TYPE ST_HMI_BASE_STATION_IN EXTENDS ST_HMI_BASE_CONTROL_IN:
STRUCT
	stButtonNavigation	: ST_HMI_BUTTON_IN;
	iStepchain			: INT; //ToDo: iStepchain HMI -> PLC STATION!?!?! (mapping missing)
	stManual			: ST_HMI_BASE_STATION_MANUAL_IN;
END_STRUCT
END_TYPE

(* stored: Version 1.1.0.1, ProductVersion 3.1.4024.11
   DUT ST_HMI_BASE_STATION_IN: Id {76fcd61e-aa0e-406e-b4eb-02a4afc93234} *)
